PROGRAM ManualLifterJog
VAR
	ArmSlowPullJogCtrlFB: MC_Jog;
END_VAR

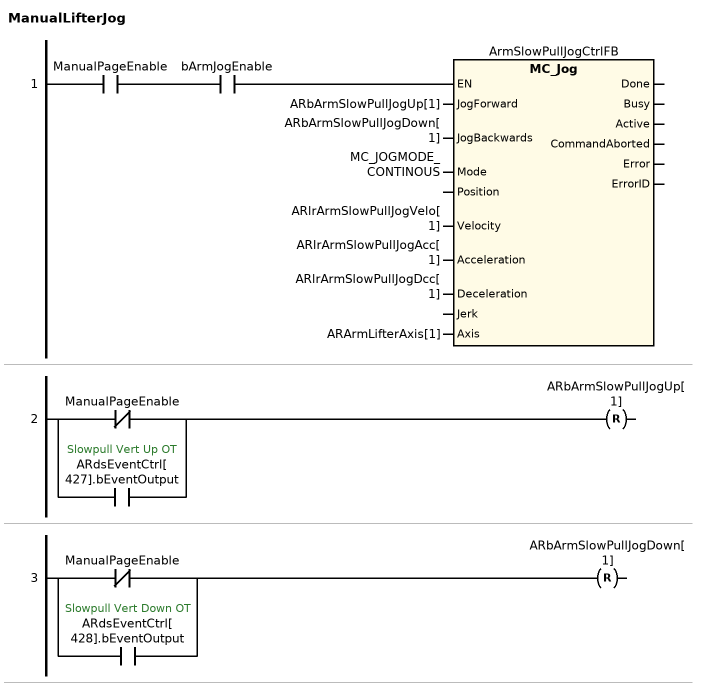
// NETWORK 1
IF ManualPageEnable AND bArmJogEnable THEN
    ArmSlowPullJogCtrlFB(
        JogForward := ARbArmSlowPullJogUp[1],
        JogBackwards := ARbArmSlowPullJogDown[1],
        Mode := MC_JOGMODE_CONTINOUS,
        Velocity := ARlrArmSlowPullJogVelo[1],
        Acceleration := ARlrArmSlowPullJogAcc[1],
        Deceleration := ARlrArmSlowPullJogDcc[1],
        Axis := ARArmLifterAxis[1]); // MC_Jog
END_IF

// NETWORK 2
//   ARdsEventCtrl[427].bEventOutput: Slowpull Vert Up OT
ARbArmSlowPullJogUp[1] R= NOT ManualPageEnable OR ARdsEventCtrl[427].bEventOutput;

// NETWORK 3
//   ARdsEventCtrl[428].bEventOutput: Slowpull Vert Down OT
ARbArmSlowPullJogDown[1] R= NOT ManualPageEnable OR ARdsEventCtrl[428].bEventOutput;

END_PROGRAM

(* stored: Version 1.1.0.1, ProductVersion 3.1.4024.12
   POU ManualLifterJog: Id {3723f729-8ac6-460f-8544-4f775736521d}, SpecialFunc None *)
